// TIA Portal V20 export
TYPE "typeCmControlNodeInterlock"
// stored: Namespace Unit1.Em4
   STRUCT
      compensator { ExternalWritable := 'False'} : "LER_typeAxisInterlock";
      feedingRoll { ExternalWritable := 'False'} : "LER_typeAxisInterlock";
      electrodeCutter { ExternalWritable := 'False'} : "LER_typeAxisInterlock";
      positionMoving { ExternalWritable := 'False'} : "LER_typeAxisInterlock";
      feederCylinder { ExternalWritable := 'False'} : "LER_typeTwoWayActuatorInterlock";
   END_STRUCT;
END_TYPE
